// Mitsubishi GX Works2 project: HB200   PLC: FX2N/FX2NC

PROGRAM MAIN
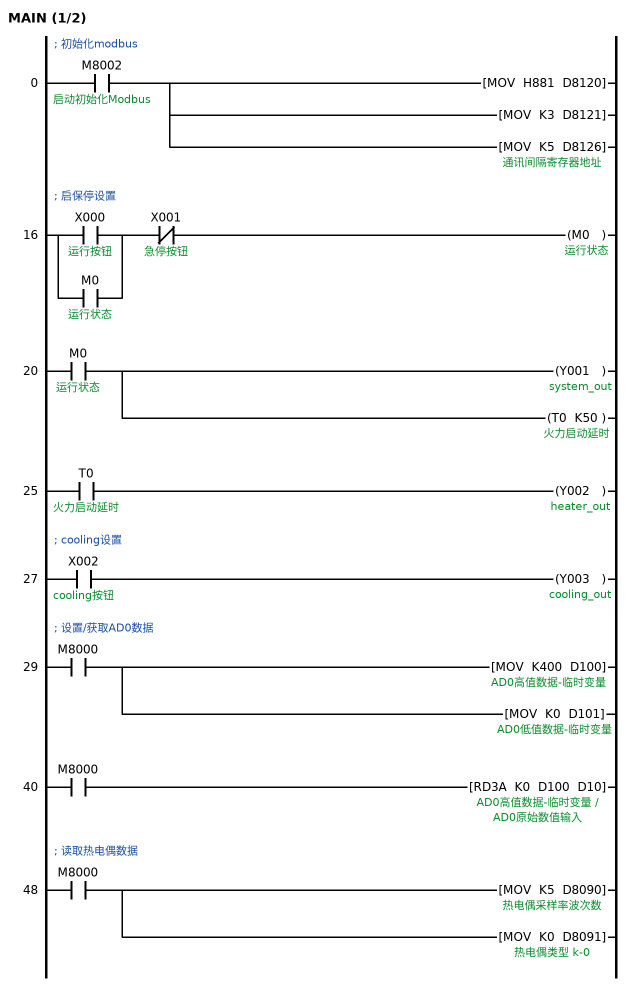
; 初始化modbus
0     LD      M8002  ; 启动初始化Modbus
      MOV     H881 D8120
        [note] MODBUS从站，9600，N，8，1
      MOV     K3 D8121
        [note] 设置站号：3
      MOV     K5 D8126  ; 通讯间隔寄存器地址
        [note] 设置通讯间隔5ms
; 启保停设置
16    LD      X000  ; 运行按钮
      OR      M0  ; 运行状态
      ANI     X001  ; 急停按钮
      OUT     M0  ; 运行状态
20    LD      M0  ; 运行状态
      OUT     Y001  ; system_out
        [note] 启动系统电量
      OUT     T0 K50  ; 火力启动延时
        [note] 延时启动5秒
25    LD      T0  ; 火力启动延时
      OUT     Y002  ; heater_out
        [note] 延时5秒后启动加热
; cooling设置
27    LD      X002  ; cooling按钮
      OUT     Y003  ; cooling_out
; 设置/获取AD0数据
29    LD      M8000
      MOV     K400 D100  ; AD0高值数据-临时变量
        [note] 设置AD0参数
      MOV     K0 D101  ; AD0低值数据-临时变量
40    LD      M8000
      RD3A    K0 D100 D10  ; AD0原始数值输入
        [note] 读取AD0数据
; 读取热电偶数据
48    LD      M8000
      MOV     K5 D8090  ; 热电偶采样率波次数
      MOV     K0 D8091  ; 热电偶类型 k-0
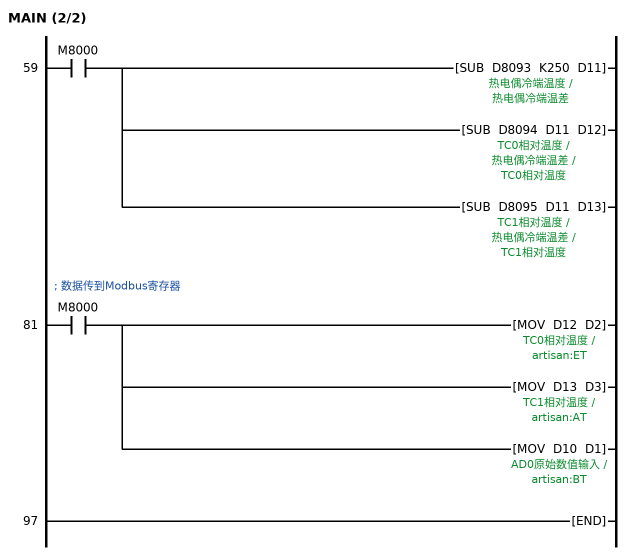
59    LD      M8000
      SUB     D8093 K250 D11  ; 热电偶冷端温度 / 热电偶冷端温差
      SUB     D8094 D11 D12  ; TC0相对温度 / TC0相对温度
      SUB     D8095 D11 D13  ; TC1相对温度 / TC1相对温度
; 数据传到Modbus寄存器
81    LD      M8000
      MOV     D12 D2  ; artisan:ET
      MOV     D13 D3  ; artisan:AT
      MOV     D10 D1  ; artisan:BT
97    END
END_PROGRAM

// device comments not shown above
M1  ; 正常运行
